FUNCTION_BLOCK TestActState2 (* CAT Function Block Type *)
  (* Standard: 61499-2 *)
  (* Version 0.0, 6/3/2026, Schneider Electric, template *)
  PACKAGE SE.Nereda;
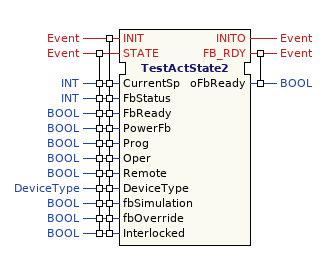
  EVENT_INPUT
    INIT WITH CurrentSp, FbStatus, Prog, Oper, Remote, FbReady, PowerFb, DeviceType, fbSimulation, fbOverride, Interlocked;
    STATE WITH CurrentSp, FbStatus, FbReady, PowerFb, Prog, Oper, Remote, DeviceType, fbSimulation, fbOverride, Interlocked;
  END_EVENT
  EVENT_OUTPUT
    INITO;
    FB_RDY WITH oFbReady;
  END_EVENT
  VAR_INPUT
    CurrentSp : INT;
    FbStatus : INT;
    FbReady : BOOL;
    PowerFb : BOOL;
    Prog : BOOL;
    Oper : BOOL;
    Remote : BOOL;
    DeviceType : DeviceType;
    fbSimulation : BOOL;
    fbOverride : BOOL;
    Interlocked : BOOL;
  END_VAR
  VAR_OUTPUT
    oFbReady : BOOL;
  END_VAR
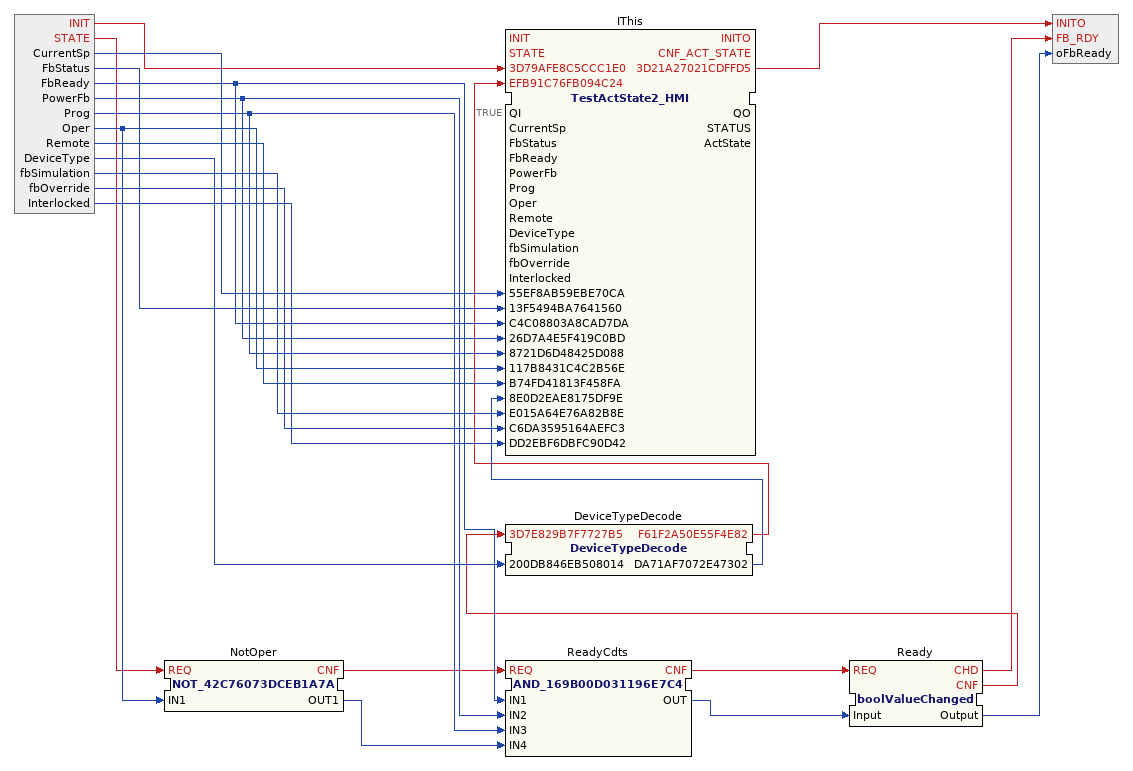
  (* Ready Conditions : Fb Ready = TRUE Fb Power = TRUE Prog = TRUE Oper = FALSE *)
  FBS
    IThis : TestActState2_HMI(QI := TRUE);
    DeviceTypeDecode : DeviceTypeDecode;
    Ready : boolValueChanged;
    ReadyCdts : AND_169B00D031196E7C4; {SET_ATTRIBUTE(Configuration.GenericFBType.InterfaceParams, Runtime.Standard#CNT:=4;OUT:BOOL)}
    NotOper : NOT_42C76073DCEB1A7A; {SET_ATTRIBUTE(Configuration.GenericFBType.InterfaceParams, Runtime.Standard#CNT:=1;OUT${CNT$}:BOOL)}
  END_FBS
  EVENT_CONNECTIONS
    Ready.CHD TO FB_RDY;
    STATE TO NotOper.REQ;
    NotOper.CNF TO ReadyCdts.REQ;
    ReadyCdts.CNF TO Ready.REQ;
    Ready.CNF TO DeviceTypeDecode.3D7E829B7F7727B5;
    INIT TO IThis.3D79AFE8C5CCC1E0;
    DeviceTypeDecode.F61F2A50E55F4E82 TO IThis.EFB91C76FB094C24;
    IThis.3D21A27021CDFFD5 TO INITO;
  END_CONNECTIONS
  DATA_CONNECTIONS
    Ready.Output TO oFbReady;
    Oper TO NotOper.IN1;
    FbReady TO ReadyCdts.IN1;
    PowerFb TO ReadyCdts.IN2;
    Prog TO ReadyCdts.IN3;
    NotOper.OUT1 TO ReadyCdts.IN4;
    ReadyCdts.OUT TO Ready.Input;
    DeviceType TO DeviceTypeDecode.200DB846EB508014;
    CurrentSp TO IThis.55EF8AB59EBE70CA;
    FbStatus TO IThis.13F5494BA7641560;
    FbReady TO IThis.C4C08803A8CAD7DA;
    PowerFb TO IThis.26D7A4E5F419C0BD;
    Prog TO IThis.8721D6D48425D088;
    Oper TO IThis.117B8431C4C2B56E;
    Remote TO IThis.B74FD41813F458FA;
    DeviceTypeDecode.DA71AF7072E47302 TO IThis.8E0D2EAE8175DF9E;
    fbSimulation TO IThis.E015A64E76A82B8E;
    fbOverride TO IThis.C6DA3595164AEFC3;
    Interlocked TO IThis.DD2EBF6DBFC90D42;
  END_CONNECTIONS
END_FUNCTION_BLOCK
